(* Schneider Machine Expert - Basic project 4pompe, file version 3.0.0.0 *)
(* ProjectInformations: Name=New project *)

HARDWARE
  Cpu 0: TM221C40R
  EthernetConfiguration: NetworkName=M221, IpAllocationMode=FixedAddress, IpAddress=0.0.0.0, SubnetMask=0.0.0.0
  SerialLineConfiguration: Baud=Baud19200, Parity=ParityEven, DataBits=DataBits8, StopBits=StopBits1, PhysicalMedium=PhysicalMediumRs485, TransmissionMode=TransmissionModeModbusRtu, SlaveId=1, Addressing=SlaveAddressing
  MastTask: UsePeriodScanMode=false, PeriodScan=100
  FastTask: Period=255
  CpuBehavior: StartingMode=StartAsPreviousState, AutoSaveRamOnEeprom=true, WatchdogPeriod=250

SYMBOLS  (address, symbol, comment, settings)
  %M0       P1_USABILE
  %M1       P2_USABILE
  %M2       P3_USABILE
  %MW0      NUM_POMPE_DA_COMANDARE
  %MW1      NUM_POMPE_MOTO
  %I0.0     LVL_MIN
  %I0.1     LVL_MAX1
  %I0.2     LVL_MAX2
  %I0.3     LVL_MAX3
  %I0.4     P1_AUTO
  %I0.5     P1_MOTO
  %I0.6     P1_ANOMALIA
  %I0.7     P2_AUTO
  %I0.8     P2_MOTO
  %I0.9     P2_ANOMALIA
  %I0.10    P3_AUTO
  %I0.11    P3_MOTO
  %I0.12    P3_ANOMALIA
  %I0.13    P4_AUTO
  %I0.14    P4_MOTO
  %I0.15    P4_ANOMALIA
  %Q0.0     P1_CMD
  %Q0.1     P2_CMD
  %Q0.2     P3_CMD
  %Q0.3     P4_CMD

POU New POU
  (* SectionNumber=1 *)

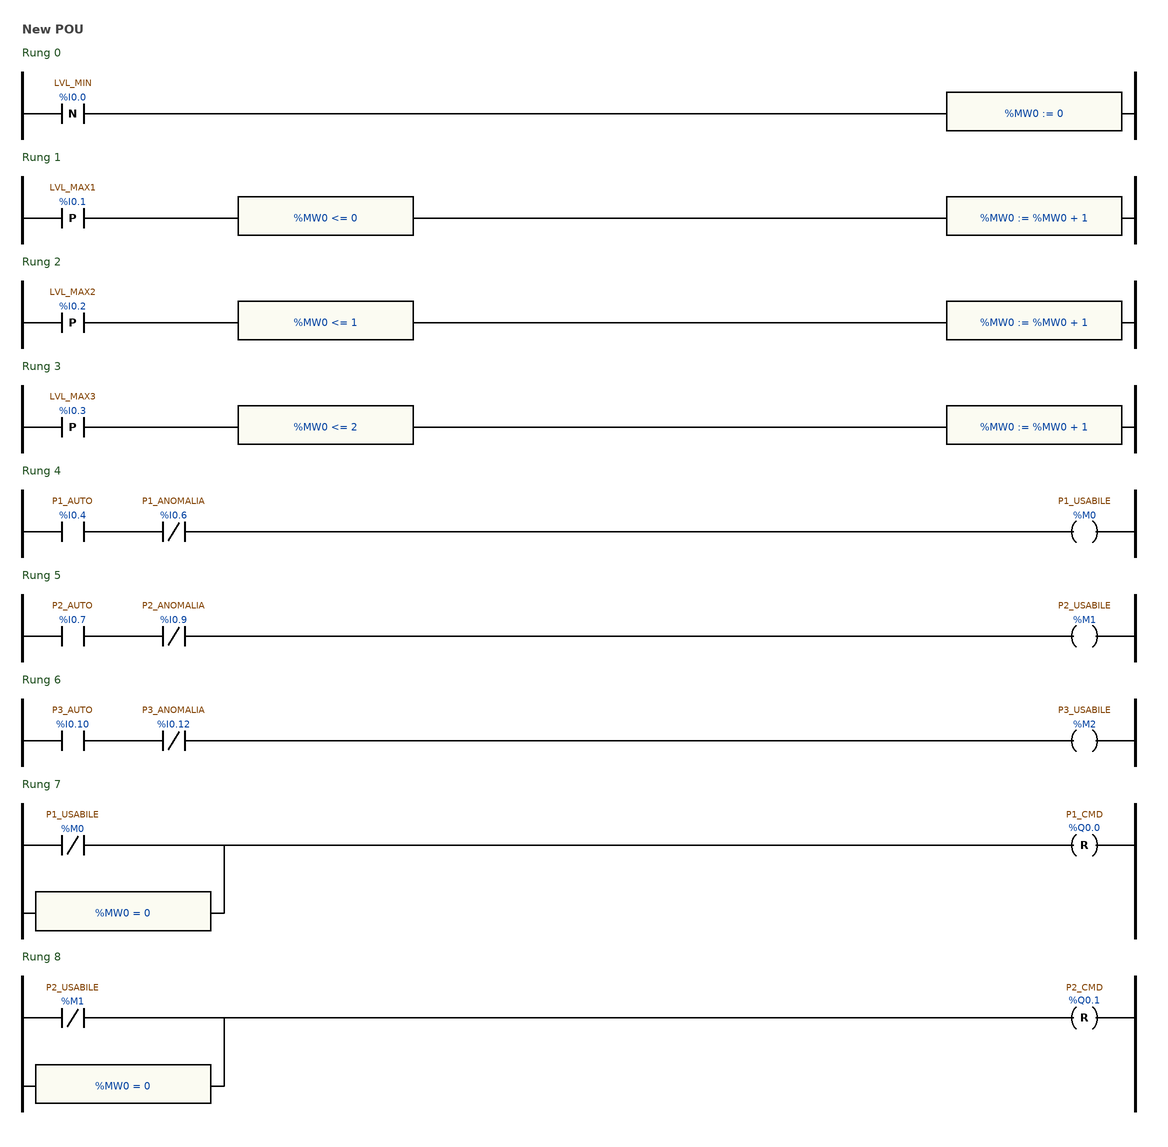

// Rung 0
  LDF %I0.0               (* LVL_MIN *)
  [ %MW0 := 0 ]           (* NUM_POMPE_DA_COMANDARE *)
  // as ST:
  //   IF FALLING(LVL_MIN) THEN NUM_POMPE_DA_COMANDARE := 0; END_IF;

// Rung 1
  LDR %I0.1               (* LVL_MAX1 *)
  AND [ %MW0 <= 0 ]       (* NUM_POMPE_DA_COMANDARE *)
  [ %MW0 := %MW0 + 1 ]    (* NUM_POMPE_DA_COMANDARE, NUM_POMPE_DA_COMANDARE *)
  // as ST:
  //   IF RISING(LVL_MAX1) AND NUM_POMPE_DA_COMANDARE <= 0 THEN NUM_POMPE_DA_COMANDARE := NUM_POMPE_DA_COMANDARE + 1; END_IF;

// Rung 2
  LDR %I0.2               (* LVL_MAX2 *)
  AND [ %MW0 <= 1 ]       (* NUM_POMPE_DA_COMANDARE *)
  [ %MW0 := %MW0 + 1 ]    (* NUM_POMPE_DA_COMANDARE, NUM_POMPE_DA_COMANDARE *)
  // as ST:
  //   IF RISING(LVL_MAX2) AND NUM_POMPE_DA_COMANDARE <= 1 THEN NUM_POMPE_DA_COMANDARE := NUM_POMPE_DA_COMANDARE + 1; END_IF;

// Rung 3
  LDR %I0.3               (* LVL_MAX3 *)
  AND [ %MW0 <= 2 ]       (* NUM_POMPE_DA_COMANDARE *)
  [ %MW0 := %MW0 + 1 ]    (* NUM_POMPE_DA_COMANDARE, NUM_POMPE_DA_COMANDARE *)
  // as ST:
  //   IF RISING(LVL_MAX3) AND NUM_POMPE_DA_COMANDARE <= 2 THEN NUM_POMPE_DA_COMANDARE := NUM_POMPE_DA_COMANDARE + 1; END_IF;

// Rung 4
  LD %I0.4                (* P1_AUTO *)
  ANDN %I0.6              (* P1_ANOMALIA *)
  ST %M0                  (* P1_USABILE *)
  // as ST:
  //   P1_USABILE := P1_AUTO AND NOT P1_ANOMALIA;

// Rung 5
  LD %I0.7                (* P2_AUTO *)
  ANDN %I0.9              (* P2_ANOMALIA *)
  ST %M1                  (* P2_USABILE *)
  // as ST:
  //   P2_USABILE := P2_AUTO AND NOT P2_ANOMALIA;

// Rung 6
  LD %I0.10               (* P3_AUTO *)
  ANDN %I0.12             (* P3_ANOMALIA *)
  ST %M2                  (* P3_USABILE *)
  // as ST:
  //   P3_USABILE := P3_AUTO AND NOT P3_ANOMALIA;

// Rung 7
  LDN %M0                 (* P1_USABILE *)
  OR [ %MW0 = 0 ]         (* NUM_POMPE_DA_COMANDARE *)
  R %Q0.0                 (* P1_CMD *)
  // as ST:
  //   IF NOT P1_USABILE OR NUM_POMPE_DA_COMANDARE = 0 THEN P1_CMD := FALSE; END_IF;

// Rung 8
  LDN %M1                 (* P2_USABILE *)
  OR [ %MW0 = 0 ]         (* NUM_POMPE_DA_COMANDARE *)
  R %Q0.1                 (* P2_CMD *)
  // as ST:
  //   IF NOT P2_USABILE OR NUM_POMPE_DA_COMANDARE = 0 THEN P2_CMD := FALSE; END_IF;

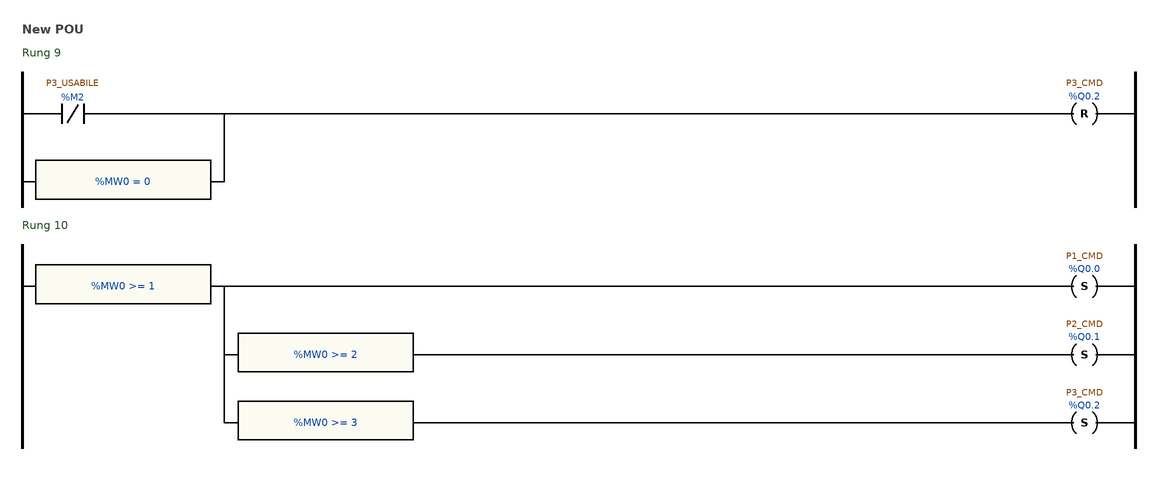

// Rung 9
  LDN %M2                 (* P3_USABILE *)
  OR [ %MW0 = 0 ]         (* NUM_POMPE_DA_COMANDARE *)
  R %Q0.2                 (* P3_CMD *)
  // as ST:
  //   IF NOT P3_USABILE OR NUM_POMPE_DA_COMANDARE = 0 THEN P3_CMD := FALSE; END_IF;

// Rung 10
  LD [ %MW0 >= 1 ]        (* NUM_POMPE_DA_COMANDARE *)
  MPS
  S %Q0.0                 (* P1_CMD *)
  MRD
  AND [ %MW0 >= 2 ]       (* NUM_POMPE_DA_COMANDARE *)
  S %Q0.1                 (* P2_CMD *)
  MPP
  AND [ %MW0 >= 3 ]       (* NUM_POMPE_DA_COMANDARE *)
  S %Q0.2                 (* P3_CMD *)
  // as ST:
  //   IF NUM_POMPE_DA_COMANDARE >= 1 THEN P1_CMD := TRUE; END_IF;
  //   IF NUM_POMPE_DA_COMANDARE >= 1 AND NUM_POMPE_DA_COMANDARE >= 2 THEN P2_CMD := TRUE; END_IF;
  //   IF NUM_POMPE_DA_COMANDARE >= 1 AND NUM_POMPE_DA_COMANDARE >= 3 THEN P3_CMD := TRUE; END_IF;
